FUNCTION_BLOCK FB_ErrorCnt
VAR_INPUT
	I_bAktiv	:BOOL;
	I_bReset	:BOOL;
END_VAR
VAR_OUTPUT
	Q_nCnt	:DINT;
END_VAR
VAR
	rtrig	:R_TRIG;
END_VAR


	rtrig(CLK:=I_bAktiv);
	IF rtrig.Q THEN
		Q_nCnt := Q_nCnt + 1;
	ELSIF I_bReset THEN
		Q_nCnt := 0;
	END_IF

END_FUNCTION_BLOCK

(* stored: Version 1.1.0.1, ProductVersion 3.1.4024.12
   POU FB_ErrorCnt: Id {3a9f1f33-9277-41d4-8480-7dfbfdc8bc62}, SpecialFunc None *)
